Staubli VAL3: advMovesEmpty.pgx

program advMovesEmpty(bool& x_bRes)
  local num l_nIndex
begin

  //return true if the advanced moves stack is empty
  x_bRes=true
  for l_nIndex=0 to size(bAdvMoveBusy)-1
    if bAdvMoveBusy[l_nIndex]
      x_bRes=false
      return
    endIf
  endFor


end
